{attribute 'GeneratedUsingTerminal: EK1100-0000-0018'}
{attribute addProperty BoxType "EK1100-0000-0018"}
{attribute addProperty Id "Beckhoff_EK12xxEK1122Beckhoff_EK12xxEK1122_F03C48A92"}
{attribute addProperty CRC "2969962182"}
{attribute addProperty Size "2"}
TYPE Beckhoff_EK12xx_B10606C6 EXTENDS EK1100_1FC0878B :
STRUCT
	{attribute addProperty Name "Beckhoff EK12xxEK1122"}
	{attribute addProperty PreviousPort "Beckhoff EK12xx : B"}
	Beckhoff_EK12xxEK1122 : Beckhoff_EK12xxEK1122_F03C48A9;
END_STRUCT
END_TYPE

(* stored: Version 1.2.0.0, ProductVersion 3.1.4024.9
   DUT Beckhoff_EK12xx_B10606C6: Id {77aad86f-592d-4f9e-bdc7-f32fe8c54b5a} *)
